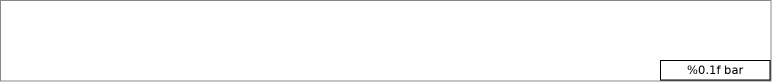
VISUALIZATION P_MAX  // 772x82
    Rectangle (660,60 110x20), "%0.1f bar", text variable: IOs_Variables.PMAX_PRESSURE_LOOSE
END_VISUALIZATION

(* stored: Version 1.1.0.1, ProductVersion 3.1.0.26
   Visu P_MAX: Id {6df48928-7a5b-4f47-a106-a8e83507c9f7} *)
